// TIA Portal V16 export
// export: Created 2023-03-29T11:04:56.4514436Z, ExportSetting WithDefaults, DisplayName Totally Integrated Automation Portal, DisplayVersion V16 Update 6, DisplayName TIA Portal Version Control Interface, DisplayVersion V16 Update 2, DisplayName TIA Portal Openness, DisplayVersion V16 Update 6, DisplayName STEP 7 Professional, DisplayVersion V16 Update 6, DisplayName STEP 7 Safety, DisplayVersion V16, DisplayName WinCC Advanced, DisplayVersion V16 Update 6
DATA_BLOCK "R_TRIG_DB_CLK"   // DB126
// stored: AutoNumber true, DBAccessibleFromOPCUA true, InstanceOfName R_TRIG, OfSystemLibElement R_TRIG, OfSystemLibVersion 1.0
"R_TRIG"
   // VAR_INPUT
   //    CLK : Bool;
   // END_VAR
   // VAR_OUTPUT
   //    Q : Bool;
   // END_VAR
   // VAR
   //    Stat_Bit : Bool;
   // END_VAR
BEGIN
END_DATA_BLOCK
